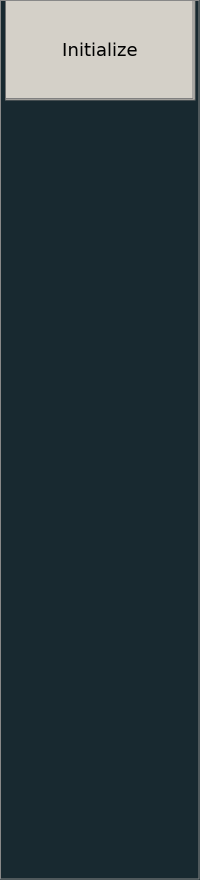
VISUALIZATION NavBarUninitialized  // 200x880
VAR_IN_OUT
	btnInitialize			: BOOL;	(*  *)
END_VAR
    Button (5,0 190x100), "Initialize"
        tap btnInitialize
END_VISUALIZATION

(* stored: Version 1.1.0.1, ProductVersion 3.1.4024.9
   Visu NavBarUninitialized: Id {60334a22-d185-410e-b47e-38542c5ab71d} *)
